(* Logix 5000 project; controller Modbus_TCP_Client_Example vendor 1 type 14 code 154 rev 32.15; software revision 32.05; part 3 of 10 *)

ADD_ON_INSTRUCTION AMP_Home_Servo   (* revision 1.0, vendor Applied Motion Products Inc. *)
// Applied Motion - Motor Homing Methods from -4  to 35  AOI
// Help:
// This AOI Execute different Homing methods from -4 to -1 and 1 to 35. Homing method -1 to -4 use for Hard Stop Homing, For all the homing methods description check the manual on Applied Motion Products Inc. website.
VAR_IN_OUT
   Input : DINT[20]; {required}   // Drive Input Assembly
        [16]   // Analog_Input1
        [4]   // Alarm_Code
        [0]   // Control_Word_Received
        [10]   // Position_Error
        [11]   // Actual_Velocity_RPS
        [12]   // Digital_Outputs
        [13]   // Digital_Inputs
        [14]   // Analog_Output1
        [15]   // Analog_Output2
        [17]   // Analog_Input2
        [18]   // Torque_Limit
        [19]   // Second_Encoder_Speed
        [1]   // OpCode1_Received
        [2]   // Control_Mode
        [3]   // Status_Code
        [5]   // Supply_Voltage
        [6]   // Applied_Torque
        [7]   // Drive_Temperature
        [8]   // Encoder_Position
        [9]   // Second_Encoder_Position
   Output : DINT[11]; {required}   // Drive Output Assembly
        [10]   // Reserved
        [4]   // Target Velocity
        [0]   // Control Word
        [3]   // Target Pos
        [1]   // OpCode 1
        [2]   // OpCode 2
        [5]   // Porifle Acceleration
        [6]   // Profile Deceleration
        [7]   // Target Torque
        [8]   // OpCode 3
        [9]   // OpCode 4
END_VAR
VAR_INPUT
   Start : BOOL; {required}   // Home the Drive (on rising edge)
   Homing_Method : DINT; {required}   // Homing Method Number Input, -4 to 35
   Home_Speed_rps : REAL; {required}   // Homing Speed 1 rps
   Home_Speed2_rps : REAL; {required}   // Homing Speed 2 rps
   Home_Acc : REAL; {required}   // Homing Acceleration of Move (rev/s/s)
   Home_Dec : REAL; {required}   // Homing Deceleration of Move (rev/s/s)
   Homing_Offset : DINT; {required}   // Homing Offset (HO) Command Value
   Hard_Stop_Homing_Torque : INT; {required}   // Homing Current (HC) Value 0-300%
END_VAR
VAR_OUTPUT
   Sent : BOOL; {access Read Only, visible}   // Home Command has been sent to drive
   In_Progress : BOOL; {access Read Only, visible}   // Homing in progress
   Done : BOOL; {access Read Only, visible}   // Homing completed without errors - Motor is Homed
   Error : BOOL; {access Read Only, visible}   // Homing failed
   State : DINT := 10; {access Read Only}   // Internal state of progress
END_VAR
VAR
   SCL_Command : INT := 'HO';   // SCL Command Characters (always 2)
   Reg2 : DINT;   // Data / SCL Register 2
   Reg1 : DINT;   // Data / SCL Register 1
   Loc_StatusCode : AMP_Status_Word_Servo; {access None}
   Loc_Input_Assembly : AMP_Input_Assembly_Servo_v2; {access None}
   Loc_Home_ONS : BOOL;
   Loc_Command_Wait2 : TIMER := (PRE := 100); {access None}   // Timer to wait between two commands
   Loc_Command_Wait1 : TIMER := (PRE := 100); {access None}   // Timer to wait between two commands
   Loc_Command_Timeout : TIMER := (PRE := 2000); {access None}   // Timer to output fault if command is not Done
   Loc_Wait_Time : TIMER := (PRE := 200); {access None}
END_VAR

ROUTINE Logic   (* ladder *)
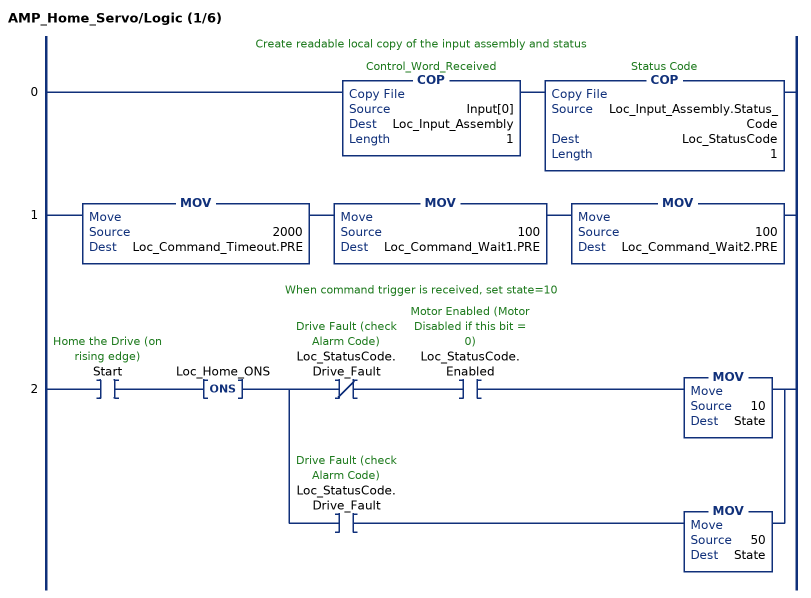
   // Create readable local copy of the input assembly and status
   0: COP(Input[0],Loc_Input_Assembly,1)COP(Loc_Input_Assembly.Status_Code,Loc_StatusCode,1);
   1: MOV(2000,Loc_Command_Timeout.PRE)MOV(100,Loc_Command_Wait1.PRE)MOV(100,Loc_Command_Wait2.PRE);
   // When command trigger is received, set state=10
   2: XIC(Start)ONS(Loc_Home_ONS)[XIO(Loc_StatusCode.Drive_Fault) XIC(Loc_StatusCode.Enabled) MOV(10,State) ,XIC(Loc_StatusCode.Drive_Fault) MOV(50,State) ];
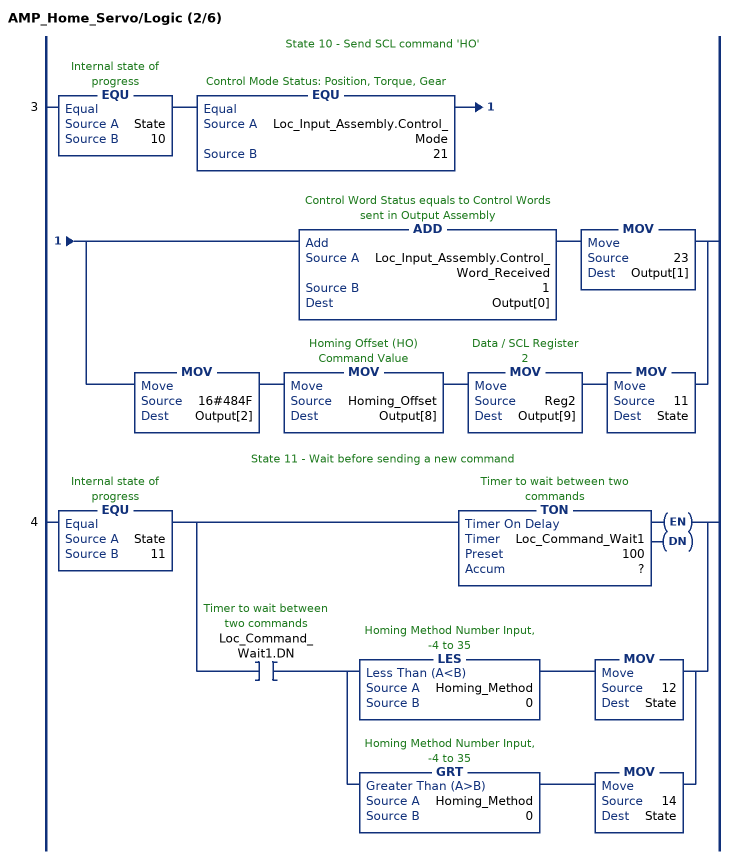
   // State 10 - Send SCL command 'HO'
   3: EQU(State,10)EQU(Loc_Input_Assembly.Control_Mode,21)[ADD(Loc_Input_Assembly.Control_Word_Received,1,Output[0]) MOV(23,Output[1]) ,MOV(16#484F,Output[2]) MOV(Homing_Offset,Output[8]) MOV(Reg2,Output[9]) MOV(11,State) ];
   // State 11 - Wait before sending a new command
   4: EQU(State,11)[TON(Loc_Command_Wait1,?,?) ,XIC(Loc_Command_Wait1.DN) [LES(Homing_Method,0) MOV(12,State) ,GRT(Homing_Method,0) MOV(14,State) ] ];
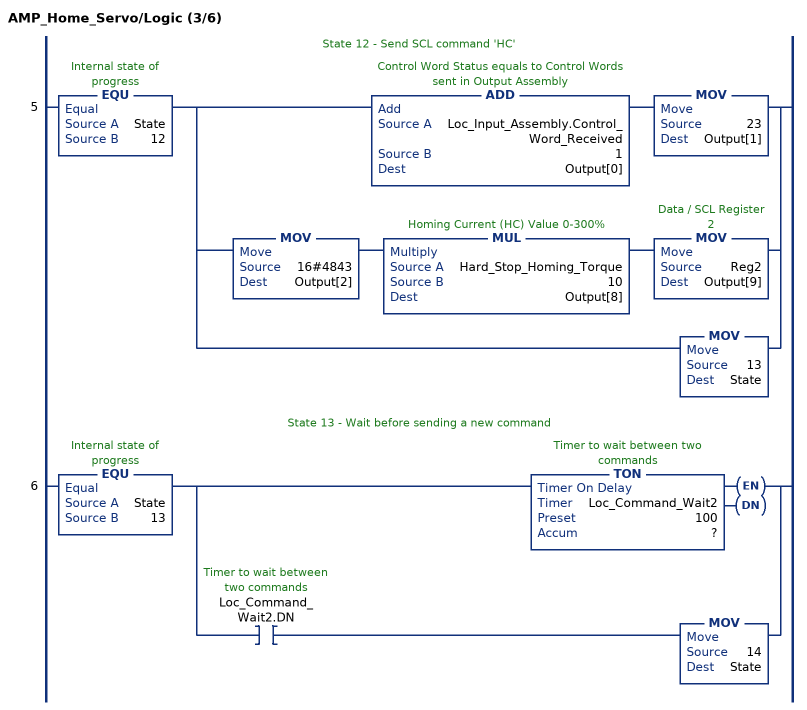
   // State 12 - Send SCL command 'HC'
   5: EQU(State,12)[ADD(Loc_Input_Assembly.Control_Word_Received,1,Output[0]) MOV(23,Output[1]) ,MOV(16#4843,Output[2]) MUL(Hard_Stop_Homing_Torque,10,Output[8]) MOV(Reg2,Output[9]) ,MOV(13,State) ];
   // State 13 - Wait before sending a new command
   6: EQU(State,13)[TON(Loc_Command_Wait2,?,?) ,XIC(Loc_Command_Wait2.DN) MOV(14,State) ];
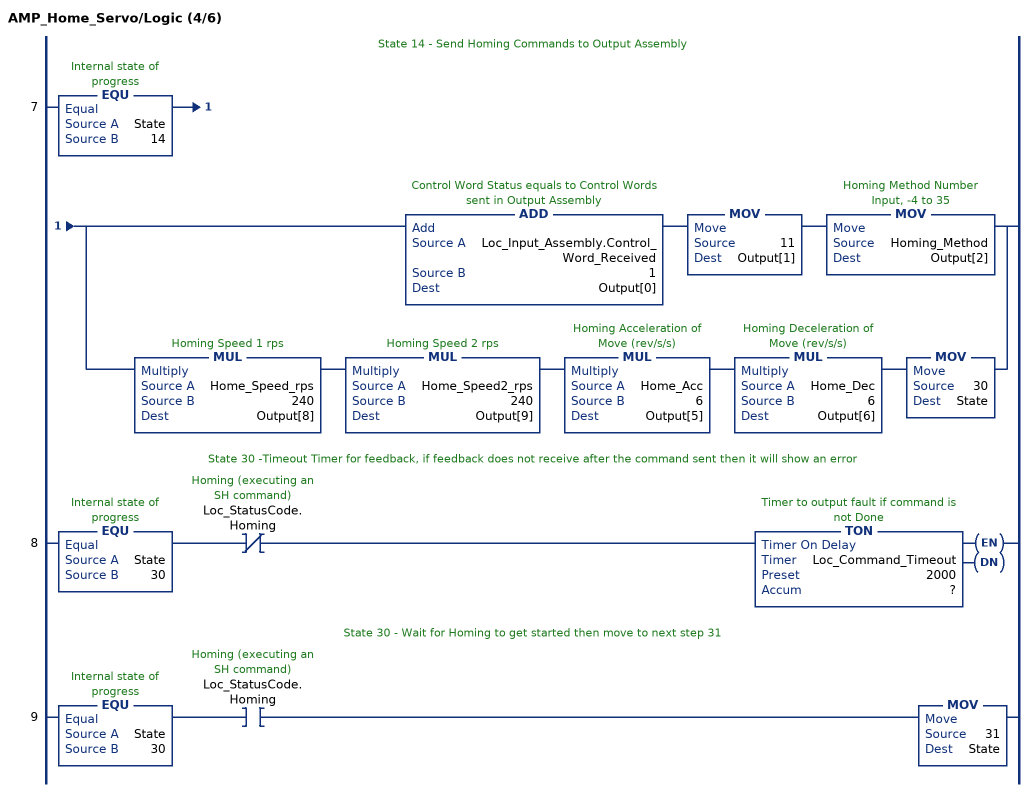
   // State 14 - Send Homing Commands to Output Assembly
   7: EQU(State,14)[ADD(Loc_Input_Assembly.Control_Word_Received,1,Output[0]) MOV(11,Output[1]) MOV(Homing_Method,Output[2]) ,MUL(Home_Speed_rps,240,Output[8]) MUL(Home_Speed2_rps,240,Output[9]) MUL(Home_Acc,6,Output[5]) MUL(Home_Dec,6,Output[6]) MOV(30,State) ];
   // State 30 -Timeout Timer for feedback, if feedback does not receive after the command sent then it will show an error
   8: EQU(State,30)XIO(Loc_StatusCode.Homing)TON(Loc_Command_Timeout,?,?);
   // State 30 - Wait for Homing to get started then move to next step 31
   9: EQU(State,30)XIC(Loc_StatusCode.Homing)MOV(31,State);
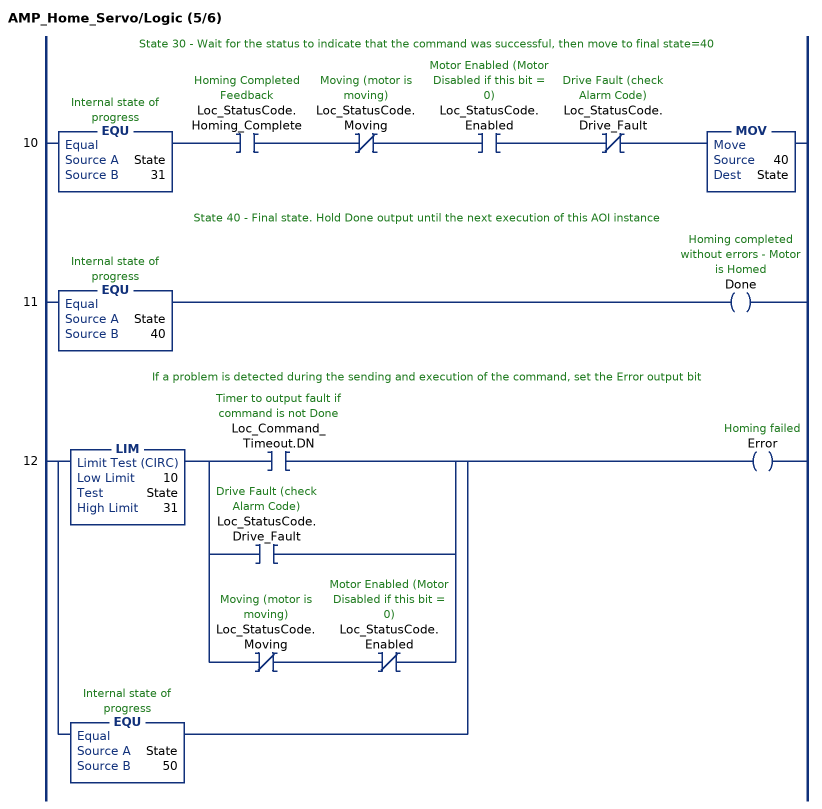
   // State 30 - Wait for the status to indicate that the command was successful, then move to final state=40
   10: EQU(State,31)XIC(Loc_StatusCode.Homing_Complete)XIO(Loc_StatusCode.Moving)XIC(Loc_StatusCode.Enabled)XIO(Loc_StatusCode.Drive_Fault)MOV(40,State);
   // State 40 - Final state. Hold Done output until the next execution of this AOI instance
   11: EQU(State,40)OTE(Done);
   // If a problem is detected during the sending and execution of the command, set the Error output bit
   12: [LIM(10,State,31) [XIC(Loc_Command_Timeout.DN) ,XIC(Loc_StatusCode.Drive_Fault) ,XIO(Loc_StatusCode.Moving) XIO(Loc_StatusCode.Enabled) ] ,EQU(State,50) ]OTE(Error);
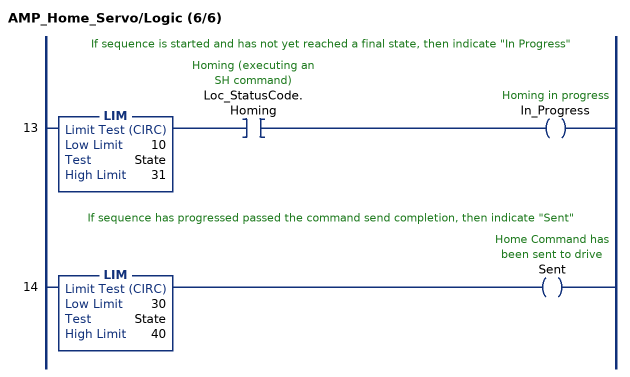
   // If sequence is started and has not yet reached a final state, then indicate "In Progress"
   13: LIM(10,State,31)XIC(Loc_StatusCode.Homing)OTE(In_Progress);
   // If sequence has progressed passed the command send completion, then indicate "Sent"
   14: LIM(30,State,40)OTE(Sent);
END_ROUTINE
END_ADD_ON_INSTRUCTION

ADD_ON_INSTRUCTION AMP_Input_Assembly   (* revision 1.0 *)
// Applied Motion - Input Assembly AOI
// Help:
// The Input Assembly AOI takes raw input data from the drive and re-interprets the data, using either scaling or copying, to appropriately named outputs.
VAR_IN_OUT
   Input : DINT[14]; {required}   // AMP_Assembly
   Output : AMP_Input_Assembly_v2; {required}
END_VAR
VAR_OUTPUT
   Status_Code : DINT; {access Read Only, visible}   // Status Code
   Alarm_Code : DINT; {access Read Only, visible}   // Alarm Code
   Voltage : REAL; {access Read Only, visible}   // Supply Voltage (V)
   Current : REAL; {access Read Only, visible}   // Actual Current (mA)
   Temp : REAL; {access Read Only, visible}   // Drive Temperature (deg C)
   Encoder_Position : DINT; {access Read Only, visible}   // Encoder Position (20,000 counts = 1 shaft turn)
   Absolute_Position : DINT; {access Read Only, visible}   // Absolute Position (20,000 counts = 1 shaft turn)
   Actual_Velocity : REAL; {access Read Only, visible}   // Actual Velocity (rev/sec, 0 when no encoder)
   Position_Error : DINT; {access Read Only, visible}
   Extended_Inputs : INT; {access Read Only, visible}   // Input Status (Extended)
   Main_Board_Inputs : INT; {access Read Only, visible}   // Input Status (Main board)
   Analog_Input_1 : DINT; {access Read Only, visible}   // Analog Input 1 (ADC counts, 0=min V, 16383 = max V)
   Analog_Input_2 : DINT; {access Read Only, visible}   // Analog Input 2 (ADC counts, 0=min V, 16383 = max V)
END_VAR
VAR
   Loc_Input_Assembly : AMP_Input_Assembly_v2; {access None}
   Loc_StatusCode : AMP_Status_Word; {access None}
END_VAR

ROUTINE Logic   (* ladder *)
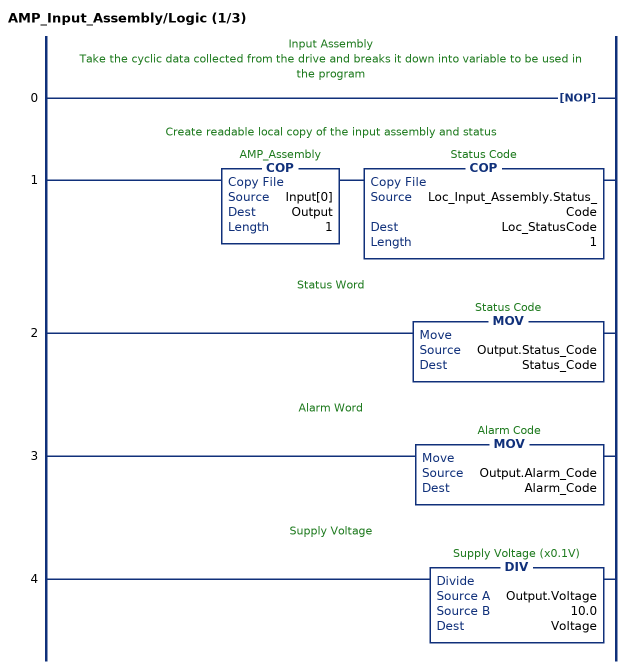
   // Input Assembly
   // Take the cyclic data collected from the drive and breaks it down into variable to be used in the program
   0: NOP();
   // Create readable local copy of the input assembly and status
   1: COP(Input[0],Output,1)COP(Loc_Input_Assembly.Status_Code,Loc_StatusCode,1);
   // Status Word
   2: MOV(Output.Status_Code,Status_Code);
   // Alarm Word
   3: MOV(Output.Alarm_Code,Alarm_Code);
   // Supply Voltage
   4: DIV(Output.Voltage,10.0,Voltage);
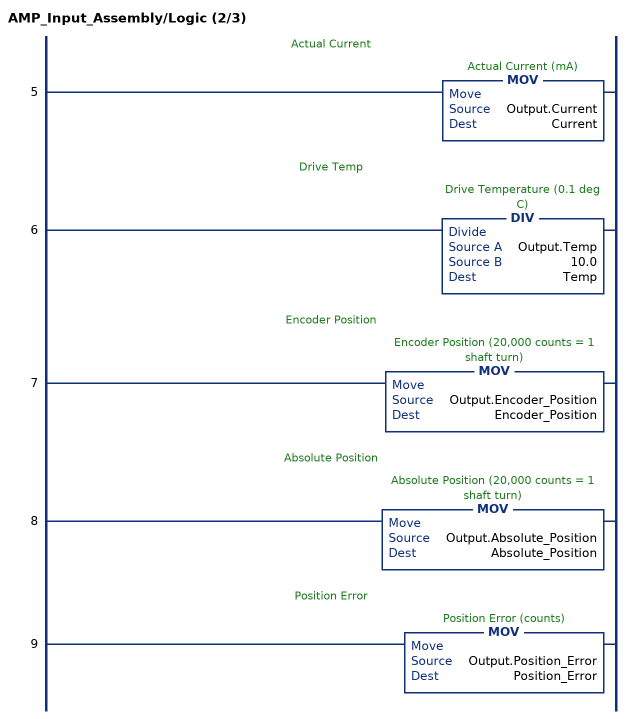
   // Actual Current
   5: MOV(Output.Current,Current);
   // Drive Temp
   6: DIV(Output.Temp,10.0,Temp);
   // Encoder Position
   7: MOV(Output.Encoder_Position,Encoder_Position);
   // Absolute Position
   8: MOV(Output.Absolute_Position,Absolute_Position);
   // Position Error
   9: MOV(Output.Position_Error,Position_Error);
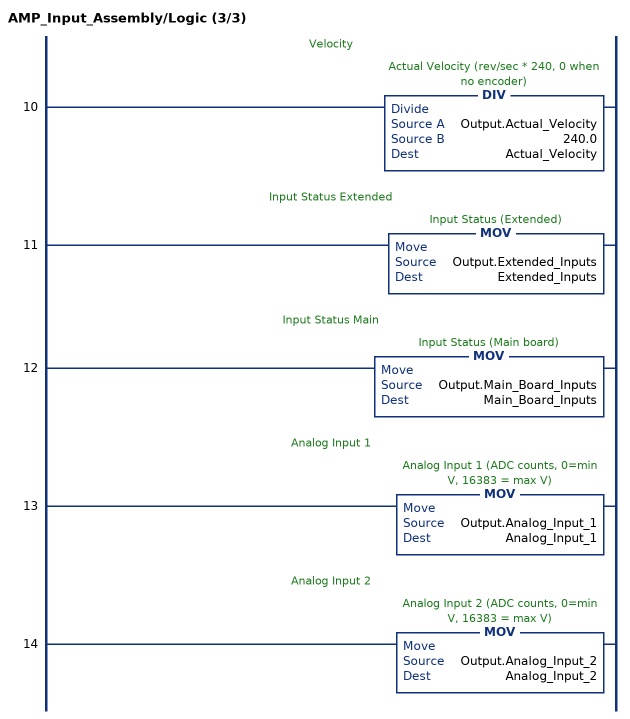
   // Velocity
   10: DIV(Output.Actual_Velocity,240.0,Actual_Velocity);
   // Input Status Extended
   11: MOV(Output.Extended_Inputs,Extended_Inputs);
   // Input Status Main
   12: MOV(Output.Main_Board_Inputs,Main_Board_Inputs);
   // Analog Input 1
   13: MOV(Output.Analog_Input_1,Analog_Input_1);
   // Analog Input 2
   14: MOV(Output.Analog_Input_2,Analog_Input_2);
END_ROUTINE
END_ADD_ON_INSTRUCTION

ADD_ON_INSTRUCTION AMP_Input_Assembly_Servo   (* revision 1.0, vendor Applied Motion Products Inc. *)
// Applied Motion - Input Assembly AOI
// Help:
// The Input Assembly AOI takes raw input data from the drive and re-interprets the data, using either scaling or copying to appropriately named outputs.
VAR_IN_OUT
   Input : DINT[20]; {required}   // AMP_Assembly
   Output : AMP_Input_Assembly_Servo_v2; {required}
END_VAR
VAR_OUTPUT
   Control_Word_Received : DINT; {access Read Only, visible}   // Control Word Status equals to Control Words sent in Output Assembly
   OpCode1_Received : DINT; {access Read Only, visible}   // OpCode 1 Status equals to OpCode1 sent in Output Assembly
   Control_Mode_Active : DINT; {visible}   // Active Control Mode (0 at startup) 1= Torque, 21= Position, 10=Velocity
   Status_Code : DINT; {access Read Only, visible}   // Status Code
   Alarm_Code : DINT; {access Read Only, visible}   // Alarm Code
   DC_Bus_Voltage : REAL; {access Read Only, visible}   // DC Bus Voltage 0.1 V: ex. 242=24.2V
   Applied_Torque_Percentage : REAL; {access Read Only, visible}   // Total Applied Torque %
   Drive_Temperature_C : REAL; {access Read Only, visible}   // Drive Temperature 0.1 deg C: ex. 305=30.5 C
   Encoder_Position : DINT; {access Read Only, visible}   // Encoder Actual Position
   Position_Error : DINT; {access Read Only, visible}   // Position Error Counts
   Actual_Velocity_rps : REAL; {access Read Only, visible}   // Actual Velocity rev/sec*2: ex. 480=2 rev/sec
   Digital_Output_Status : INT; {access Read Only, visible}   // Digital Output Status
   Digital_Input_Status : INT; {access Read Only, visible}   // Digital Input Status
   Analog_Output1 : DINT; {visible}   // Analog Output 1 Value
   Analog_Output2 : DINT; {visible}   // Analog Output 2 Value
   Analog_Input_1 : DINT; {access Read Only, visible}   // Analog Input 1 Value
   Analog_Input_2 : DINT; {access Read Only, visible}   // Analog Input 2 Value
   Torque_Limit : DINT; {visible}   // Torque Limit Set Point Feedback
   External_Encoder_Position : DINT; {access Read Only, visible}   // External Encoder Position (for full closed loop servo only)
   External_Encoder_Speed_rps : DINT; {visible}   // External Encoder Speed(for full closed loop servo only)
END_VAR
VAR
   Loc_StatusCode : AMP_Status_Word_Servo; {access None}
   Loc_Input_Assembly : AMP_Input_Assembly_Servo_v2; {access None}
END_VAR

ROUTINE Logic   (* ladder *)
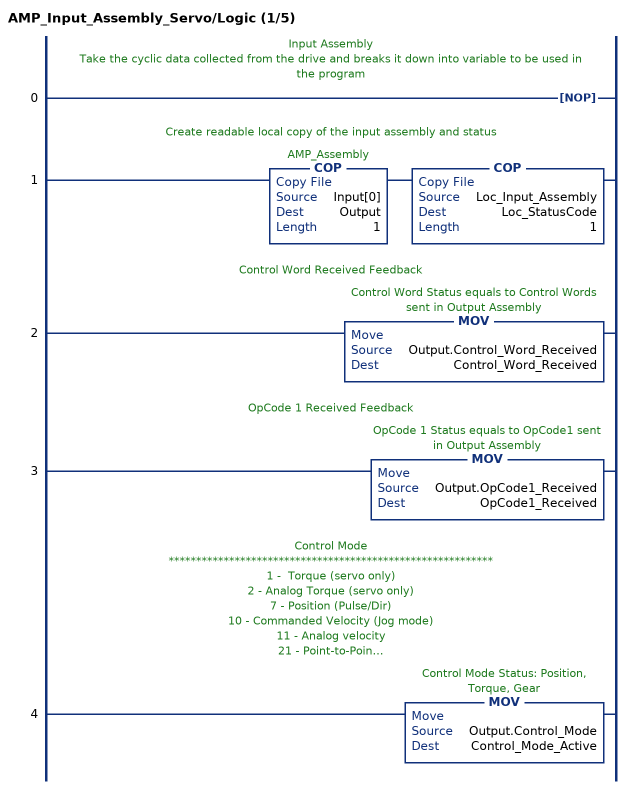
   // Input Assembly
   // Take the cyclic data collected from the drive and breaks it down into variable to be used in the program
   0: NOP();
   // Create readable local copy of the input assembly and status
   1: COP(Input[0],Output,1)COP(Loc_Input_Assembly,Loc_StatusCode,1);
   // Control Word Received Feedback
   2: MOV(Output.Control_Word_Received,Control_Word_Received);
   // OpCode 1 Received Feedback
   3: MOV(Output.OpCode1_Received,OpCode1_Received);
   // Control Mode
   // ***********************************************************
   //  1 -  Torque (servo only)
   // 2 - Analog Torque (servo only)
   // 7 - Position (Pulse/Dir)
   // 10 - Commanded Velocity (Jog mode)
   // 11 - Analog velocity
   // 21 - Point-to-Point
   // 22 - Analog Position
   4: MOV(Output.Control_Mode,Control_Mode_Active);
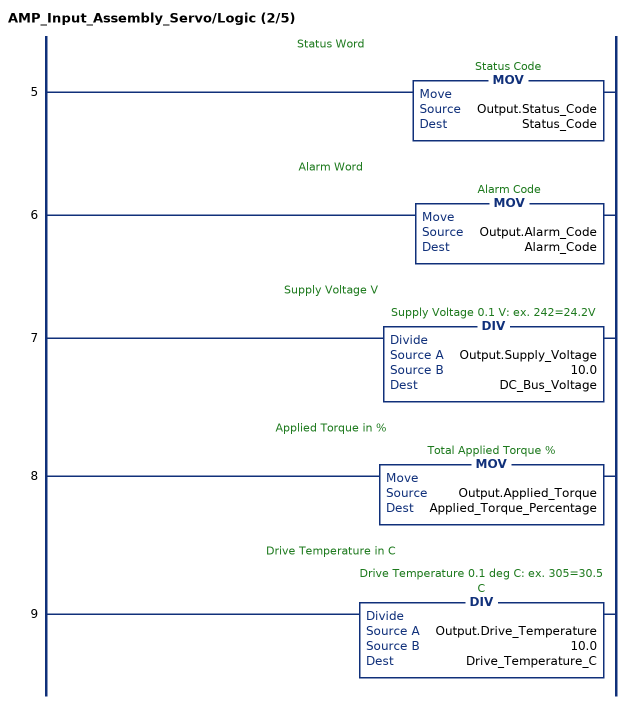
   // Status Word
   5: MOV(Output.Status_Code,Status_Code);
   // Alarm Word
   6: MOV(Output.Alarm_Code,Alarm_Code);
   // Supply Voltage V
   7: DIV(Output.Supply_Voltage,10.0,DC_Bus_Voltage);
   // Applied Torque in %
   8: MOV(Output.Applied_Torque,Applied_Torque_Percentage);
   // Drive Temperature in C
   9: DIV(Output.Drive_Temperature,10.0,Drive_Temperature_C);
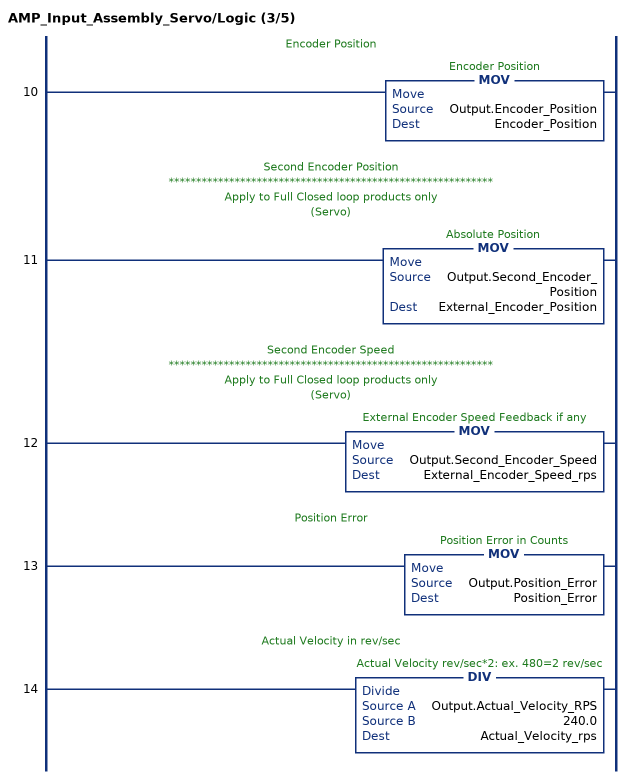
   // Encoder Position
   10: MOV(Output.Encoder_Position,Encoder_Position);
   // Second Encoder Position
   // ***********************************************************
   // Apply to Full Closed loop products only
   // (Servo)
   11: MOV(Output.Second_Encoder_Position,External_Encoder_Position);
   // Second Encoder Speed
   // ***********************************************************
   // Apply to Full Closed loop products only
   // (Servo)
   12: MOV(Output.Second_Encoder_Speed,External_Encoder_Speed_rps);
   // Position Error
   13: MOV(Output.Position_Error,Position_Error);
   // Actual Velocity in rev/sec
   14: DIV(Output.Actual_Velocity_RPS,240.0,Actual_Velocity_rps);
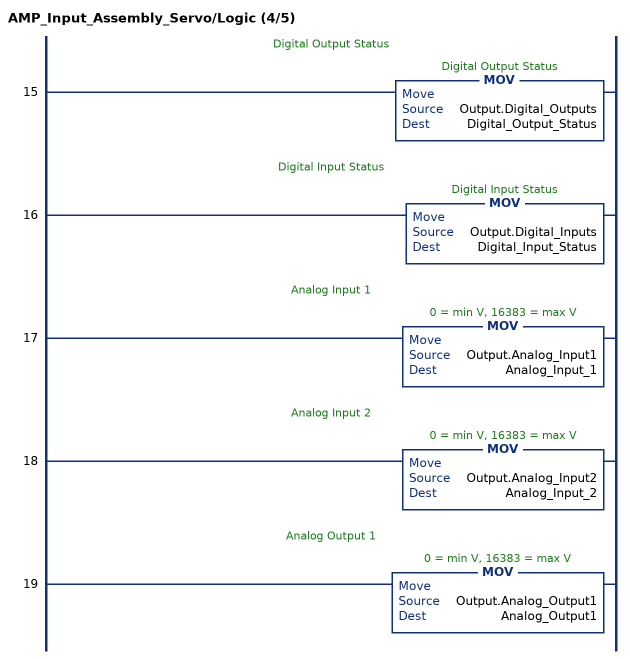
   // Digital Output Status
   15: MOV(Output.Digital_Outputs,Digital_Output_Status);
   // Digital Input Status
   16: MOV(Output.Digital_Inputs,Digital_Input_Status);
   // Analog Input 1
   17: MOV(Output.Analog_Input1,Analog_Input_1);
   // Analog Input 2
   18: MOV(Output.Analog_Input2,Analog_Input_2);
   // Analog Output 1
   19: MOV(Output.Analog_Output1,Analog_Output1);
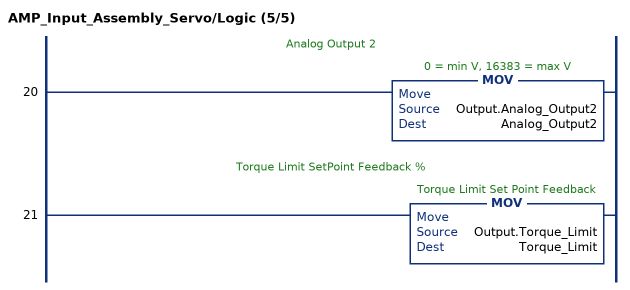
   // Analog Output 2
   20: MOV(Output.Analog_Output2,Analog_Output2);
   // Torque Limit SetPoint Feedback %
   21: MOV(Output.Torque_Limit,Torque_Limit);
END_ROUTINE
END_ADD_ON_INSTRUCTION

ADD_ON_INSTRUCTION AMP_Jog_Move   (* revision 1.0 *)
// Applied Motion - Jog Move AOI
// Help:
// The Jog Move AOI is used to start jogging an axis at a specified speed and direction (a negative speed set point implies a CCW direction).
VAR_IN_OUT
   Input : DINT[14]; {required}   // Drive Input Assembly
   Output : DINT[16]; {required}   // Drive Output Assembly
        [0]   // Command Word
        [10]   // Data/Register 1
        [11]   // Data/Register 2
        [1]   // Jog Speed (0.25 rev/min)
        [2]   // Jog Acceleration (10 rev/s/s)
        [3]   // Jog Deceleration (10 rev/s/s)
        [4]   // Point-to-Point Velocity (0.25 rev/min)
        [5]   // Point-to-Point Acceleration (10 rev/min/s)
        [6]   // Point-to-Point Deceleration (10 rev/min/s)
        [7]   // Point-to-Point Distance (Motor steps)
        [9]   // (2x ASCII Letters in 16 lower word)
END_VAR
VAR_INPUT
   RPI : DINT := 100; {visible}   // Drive Connection Request Packet Interval (milliseconds)
   Start : BOOL; {required}   // Start the Relative Move
   Speed : REAL; {required}   // Velocity of Move (rev/min)
   Acc : REAL; {required}   // Acceleration of Move (rev/s/s)
   Dec : REAL; {required}   // Deceleration (rev/s/s)
END_VAR
VAR_OUTPUT
   Sent : BOOL; {access Read Only, visible}   // Move has been sent to drive
   In_Progress : BOOL; {access Read Only, visible}   // Move in progress
   Done : BOOL; {access Read Only, visible}   // Move completed without errors - desired position reached
   Error : BOOL; {access Read Only, visible}   // Move failed to complete - drive not ready or faulted
   State : DINT := 10; {access Read Only}   // Internal state of progress
END_VAR
VAR
   Loc_StatusCode : AMP_Status_Word;
   Loc_CommandOff_Timer : TIMER;   // Timer to make sure command value was 0 before sending a new command
   Loc_CommandOn_Timer : TIMER;   // Timer to make sure command value is set long enough to be sent to drive
   Loc_Input_Assembly : AMP_Input_Assembly_v2; {access None}
   Loc_Start_ONS : BOOL; {access None}
   Loc_AlarmCode : AMP_Alarm_Word; {access None}
END_VAR

ROUTINE Logic   (* ladder *)
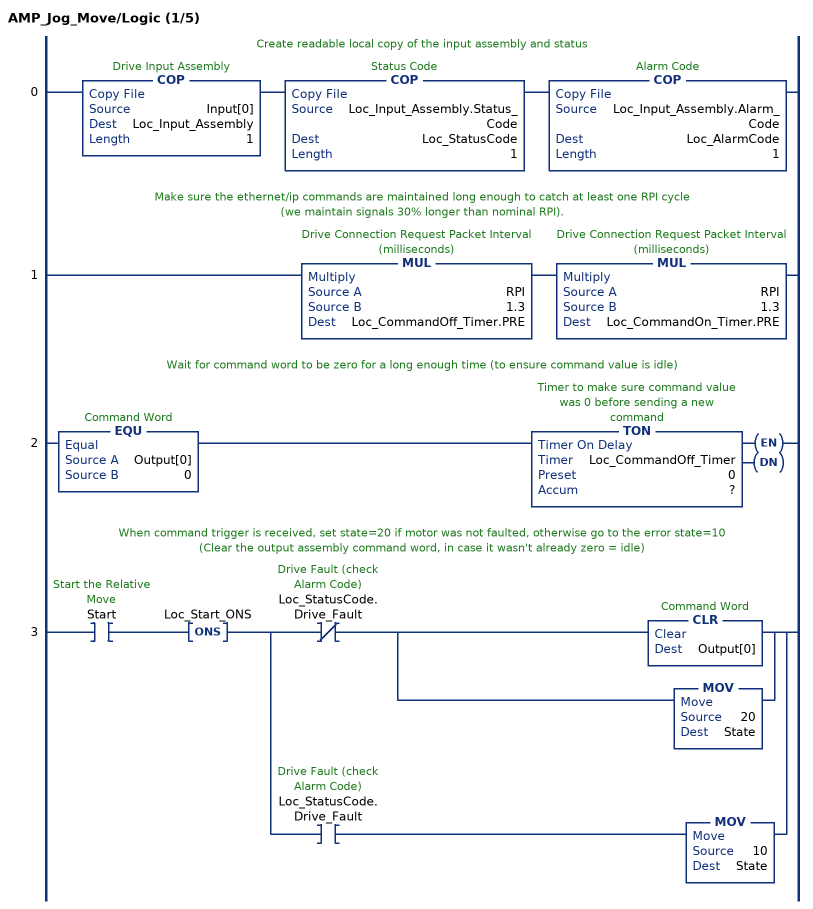
   // Create readable local copy of the input assembly and status
   0: COP(Input[0],Loc_Input_Assembly,1)COP(Loc_Input_Assembly.Status_Code,Loc_StatusCode,1)COP(Loc_Input_Assembly.Alarm_Code,Loc_AlarmCode,1);
   // Make sure the ethernet/ip commands are maintained long enough to catch at least one RPI cycle
   // (we maintain signals 30% longer than nominal RPI).
   1: MUL(RPI,1.3,Loc_CommandOff_Timer.PRE)MUL(RPI,1.3,Loc_CommandOn_Timer.PRE);
   // Wait for command word to be zero for a long enough time (to ensure command value is idle)
   2: EQU(Output[0],0)TON(Loc_CommandOff_Timer,?,?);
   // When command trigger is received, set state=20 if motor was not faulted, otherwise go to the error state=10
   // (Clear the output assembly command word, in case it wasn't already zero = idle)
   3: XIC(Start)ONS(Loc_Start_ONS)[XIO(Loc_StatusCode.Drive_Fault) [CLR(Output[0]) ,MOV(20,State) ] ,XIC(Loc_StatusCode.Drive_Fault) MOV(10,State) ];
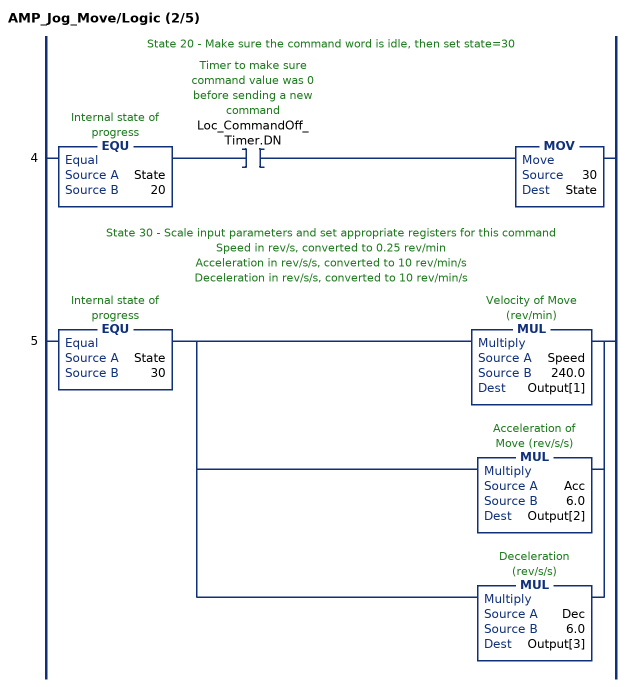
   // State 20 - Make sure the command word is idle, then set state=30
   4: EQU(State,20)XIC(Loc_CommandOff_Timer.DN)MOV(30,State);
   // State 30 - Scale input parameters and set appropriate registers for this command
   // Speed in rev/s, converted to 0.25 rev/min
   // Acceleration in rev/s/s, converted to 10 rev/min/s
   // Deceleration in rev/s/s, converted to 10 rev/min/s
   5: EQU(State,30)[MUL(Speed,240.0,Output[1]) ,MUL(Acc,6.0,Output[2]) ,MUL(Dec,6.0,Output[3]) ];
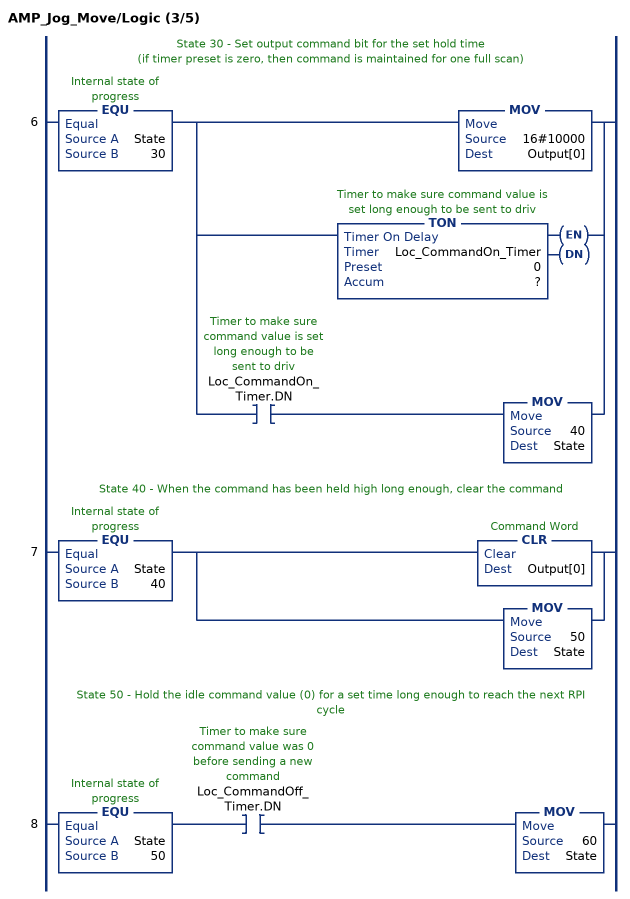
   // State 30 - Set output command bit for the set hold time
   // (if timer preset is zero, then command is maintained for one full scan)
   6: EQU(State,30)[MOV(16#10000,Output[0]) ,TON(Loc_CommandOn_Timer,?,?) ,XIC(Loc_CommandOn_Timer.DN) MOV(40,State) ];
   // State 40 - When the command has been held high long enough, clear the command
   7: EQU(State,40)[CLR(Output[0]) ,MOV(50,State) ];
   // State 50 - Hold the idle command value (0) for a set time long enough to reach the next RPI cycle
   8: EQU(State,50)XIC(Loc_CommandOff_Timer.DN)MOV(60,State);
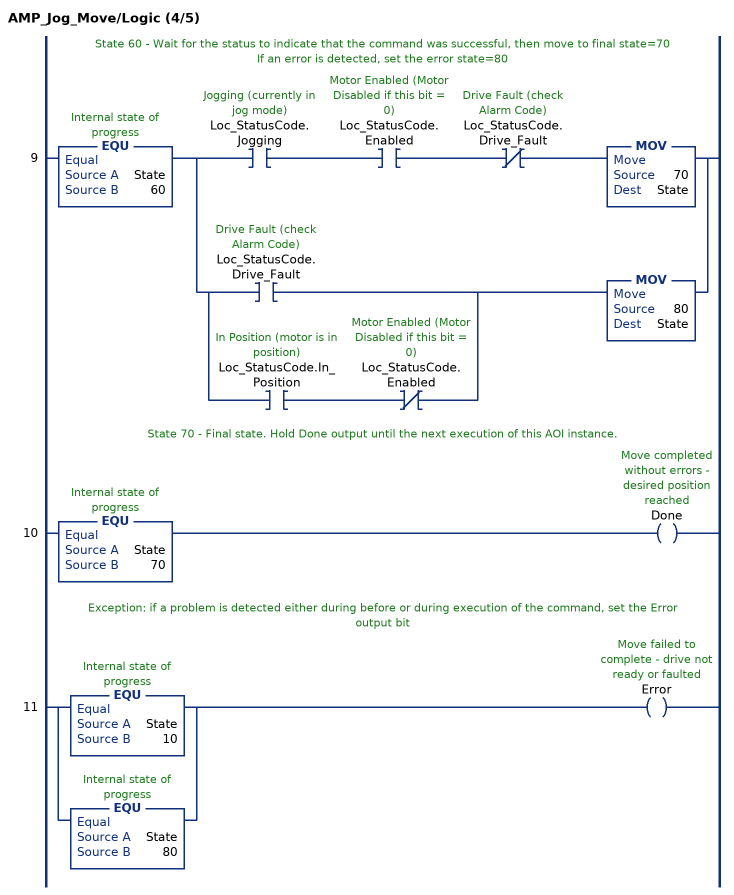
   // State 60 - Wait for the status to indicate that the command was successful, then move to final state=70
   // If an error is detected, set the error state=80
   9: EQU(State,60)[XIC(Loc_StatusCode.Jogging) XIC(Loc_StatusCode.Enabled) XIO(Loc_StatusCode.Drive_Fault) MOV(70,State) ,[XIC(Loc_StatusCode.Drive_Fault) ,XIC(Loc_StatusCode.In_Position) XIO(Loc_StatusCode.Enabled) ] MOV(80,State) ];
   // State 70 - Final state. Hold Done output until the next execution of this AOI instance.
   10: EQU(State,70)OTE(Done);
   // Exception: if a problem is detected either during before or during execution of the command, set the Error output bit
   11: [EQU(State,10) ,EQU(State,80) ]OTE(Error);
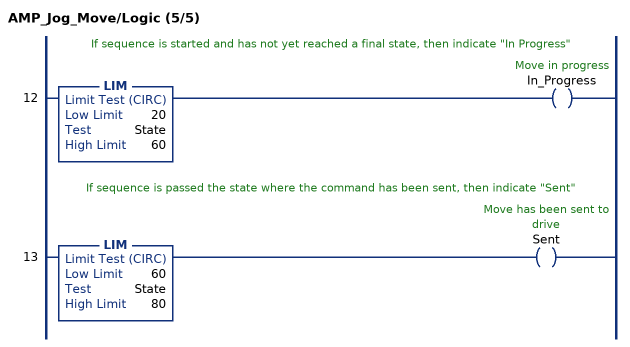
   // If sequence is started and has not yet reached a final state, then indicate "In Progress"
   12: LIM(20,State,60)OTE(In_Progress);
   // If sequence is passed the state where the command has been sent, then indicate "Sent"
   13: LIM(60,State,80)OTE(Sent);
END_ROUTINE
END_ADD_ON_INSTRUCTION
